TYPE Tabs_Tabs_other :
STRUCT
END_STRUCT
END_TYPE

(* stored: Version 1.1.0.1, ProductVersion 3.1.4024.9
   DUT Tabs_Tabs_other: Id {e173d4c7-b457-44c2-af9e-dd02427a3626} *)
